TYPE ST_Configuration :
STRUCT
  PortalConfig        : ST_CONFIG_PORTAL;
  JobConfig           : ST_CONFIG_JOBS;
END_STRUCT
END_TYPE

(* stored: Version 1.1.0.1
   DUT ST_Configuration: Id {751e9be0-0116-4a27-b9d5-2088d21242fd} *)
